ABB RobotStudio station: VRM_Team_Project_JM_VS_BP.rspag

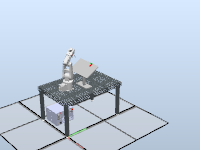
--- station ---
Station VRM_project_drawing (saved by RobotStudio 20.4.9280.0)
Controller Controller1, task T_ROB1: task frame (RAPID world) sits at (-420.14, 370.5, 830) mm, rotated rx 0 ry 0 rz 90 deg in the station
Controller Controller1
  mechanical unit ROB_1: IRB120_3_58__01, 6 joints, base frame (0, 0, 0) mm
Layout (positions relative to the parent item):
  - IRB120_3_58__01 [mechanism, from Robots\IRB120_3_58_G_01.rslib] at (-420.14, 370.5, 830) mm, rotated rx 0 ry 0 rz 90 deg; joint values [0.5236, 0, -0.5236, 0, 1.5708, 1.5708] (rad or m)
  - TraceTCP [smart component, from Components\TraceTCP.rslib]
      properties: Robot=IRB120_3_58__01
  - Assembly_all_test [part, from Libraries\Assembly_all_test.rslib] at (-451.59, -1823, 792.9) mm, rotated rx 90 ry 0 rz 180 deg
  - pen_gripper [mechanism] at (-551.41, 597.87, 1539.27) mm, rotated rx 150 ry 0 rz -150 deg
      TCP pen_gripper at (59.5, 0, 34.55) mm, rotated rx 0 ry 90 rz 0 deg
      links: Gripper_VS_JM_PB_2
  - fix [part] at (-536.37, 640.91, 1487.74) mm, rotated rx 150 ry 0 rz -150 deg
  - stul (1) [part] at (-632.9, 571.47, 830) mm
  - IRC5_Compact [part, from Equipment\IRC5_Compact__02.rslib] at (-476.14, 69.39, 0) mm, rotated rx 0 ry 0 rz 90 deg
Attachment: pen_gripper is attached to IRB120_3_58__01 / Link6
Attachment: fix is attached to pen_gripper / Gripper_VS_JM_PB_2
Station logic (signal -> signal, property => property):
  Controller1.DO_draw -> TraceTCP.Enabled
Targets, tools, work objects and paths stored in the station and not in the controller backup, written as RAPID:
! task T_ROB1
MODULE Module1
  PROC Path_10()
    MoveJ draw,v1000,z100,pen_gripper\WObj:=drawing;
  ENDPROC
ENDMODULE


--- Backups/Controller1/RAPID/TASK1/PROGMOD/CalibData.mod ---
MODULE CalibData
    PERS tooldata Pen_TCP:=[TRUE,[[110,0,140],[0.707106781,0,0.707106781,0]],[1,[10.7435139,0,140],[1,0,0,0],0,0,0]];
    PERS wobjdata drawing:=[FALSE,TRUE,"",[[479.496,-215.388859997,488.169267438],[0.257638751,0,0.966241312,0]],[[0,0,0],[1,0,0,0]]];

   ! PERS tooldata pen_gripper:=[TRUE,[[-34.55,0,59.5],[1,0,0,0]],[1,[-6.586,-0.006,22.601],[1,0,0,0],0,0,0]];
     PERS tooldata pen_gripper:=[TRUE,[[-34.55,0,146],[1,0,0,0]],[1,[-6.586,-0.006,22.601],[1,0,0,0],0,0,0]];
ENDMODULE

--- Backups/Controller1/RAPID/TASK1/PROGMOD/Module1.mod ---
MODULE Module1
        VAR robtarget Point;
        CONST jointtarget HOME:=[[30,0,-30,0,90,90],[9E+09,9E+09,9E+09,9E+09,9E+09,9E+09]];

        VAR num x_num{2000};
        VAR num y_num{2000};
        VAR num states{2000};
        VAR num count := 1;
        VAR num START := 0;
        VAR num new_path := 0;
        VAR num x_start :=0;
        VAR num y_start :=0;
        !CONST num pen_offs := -86.5;

        VAR speeddata speed := v500;
        VAR zonedata zone := fine;

    CONST robtarget draw:=[[0,0,0],[1,0,0,0],[-1,0,-1,0],[9E+09,9E+09,9E+09,9E+09,9E+09,9E+09]];

    PROC main()

        SetDO DO_draw,0;
        MoveAbsJ HOME,v500,z100,pen_gripper\WObj:=drawing;

        IF START = 1 THEN

            SetDO DO_draw,0;
            MoveJ draw,v500,z10,pen_gripper\WObj:=drawing;

        FOR i FROM 1 TO count DO

            IF states{i} = 1 THEN

                IF new_path = 0 THEN

                    x_start := x_num{i};
                    y_start := y_num{i};
                    new_path := 1;

                ENDIF

            ELSEIF states{i} = 2 THEN

                MoveL Offs(draw,x_start,y_start,-5),speed,zone,pen_gripper\WObj:=drawing;

                MoveL Offs(draw,x_start,y_start,0),speed,zone,pen_gripper\WObj:=drawing;
                SetDO DO_draw,1;

                MoveL Offs(draw,x_num{i},y_num{i},0),speed,zone,pen_gripper\WObj:=drawing;
                SetDO DO_draw,0;

                MoveL Offs(draw,x_num{i},y_num{i},-5),speed,zone,pen_gripper\WObj:=drawing;
                new_path :=0;

            ELSEIF states{i} = 3 THEN

                MoveL Offs(draw,x_num{i},y_num{i},-5),speed,zone,pen_gripper\WObj:=drawing;

                MoveL Offs(draw,x_num{i},y_num{i},0),speed,zone,pen_gripper\WObj:=drawing;
                SetDO DO_draw,1;

                MoveL Offs(draw,x_num{i},y_num{i},-5),speed,zone,pen_gripper\WObj:=drawing;
                SetDO DO_draw,0;

                new_path :=0;

            ENDIF
        ENDFOR

        MoveAbsJ HOME,v500,z100,pen_gripper\WObj:=drawing;
        START := 0;

        ENDIF

    ENDPROC

ENDMODULE

--- Backups/Controller1/SYSPAR/EIO.cfg ---
EIO:CFG_1.0:6:1::
#
EIO_SIGNAL:

      -Name "DO_draw" -SignalType "DO"
